// TIA Portal V20 export
DATA_BLOCK "HmiInterface"   // DB13
// stored: Access Published, MemoryReserve 100, Namespace Unit1
   VAR
      AutoStartEnable : Bool;
      InitializeEnable : Bool;
      PartData : Array[0..18] of "LER_typePartData";
      partDataSave : Bool;
      partDataClear : Bool;
      partDataAllClear : Bool;
      partDataSelect : Int;
      allBrakeTest : "LER_typeBrakeTestUnitInterface";
   END_VAR
   VAR RETAIN
      cmFFU : "LER_typeLIU117Interface";
      FFU_SleepModeRunPct : Real;
   END_VAR
   VAR
      "========Communication========" : Bool;
   END_VAR
   VAR RETAIN
      BA030 : "LER_typeCommunicationInterface";
      BA040 : "LER_typeCommunicationInterface";
   END_VAR
   VAR
      StackRnRPopup : Bool;
   END_VAR
BEGIN
END_DATA_BLOCK
